FUNCTION_BLOCK ConfigurationManagerC
  (* Standard: 61499-2 *)
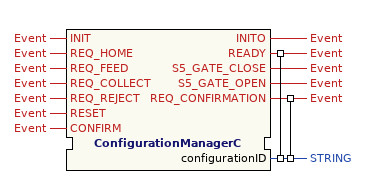
  EVENT_INPUT
    INIT;
    REQ_HOME;
    REQ_FEED;
    REQ_COLLECT;
    REQ_REJECT;
    RESET;
    CONFIRM;
  END_EVENT
  EVENT_OUTPUT
    INITO;
    READY WITH configurationID;
    S5_GATE_CLOSE;
    S5_GATE_OPEN;
    REQ_CONFIRMATION WITH configurationID;
  END_EVENT
  VAR_OUTPUT
    configurationID : STRING;
  END_VAR
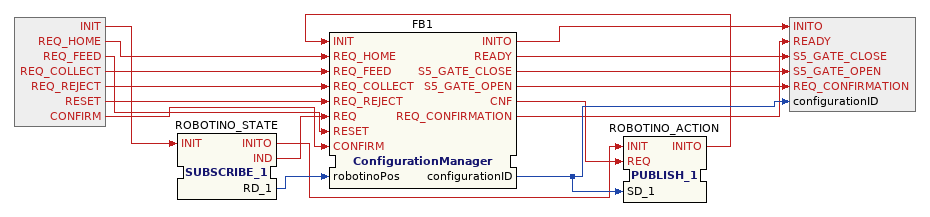
  FBS
    FB1 : ConfigurationManager;
    ROBOTINO_ACTION : PUBLISH_1;
    ROBOTINO_STATE : SUBSCRIBE_1;
  END_FBS
  EVENT_CONNECTIONS
    REQ_HOME TO FB1.REQ_HOME;
    REQ_FEED TO FB1.REQ_FEED;
    REQ_COLLECT TO FB1.REQ_COLLECT;
    REQ_REJECT TO FB1.REQ_REJECT;
    FB1.INITO TO INITO;
    FB1.READY TO READY;
    FB1.S5_GATE_CLOSE TO S5_GATE_CLOSE;
    FB1.S5_GATE_OPEN TO S5_GATE_OPEN;
    ROBOTINO_ACTION.INITO TO FB1.INIT;
    INIT TO ROBOTINO_STATE.INIT;
    RESET TO FB1.RESET;
    FB1.REQ_CONFIRMATION TO REQ_CONFIRMATION;
    CONFIRM TO FB1.CONFIRM;
    ROBOTINO_STATE.INITO TO ROBOTINO_ACTION.INIT;
    ROBOTINO_STATE.IND TO FB1.REQ;
    FB1.CNF TO ROBOTINO_ACTION.REQ;
  END_CONNECTIONS
  DATA_CONNECTIONS
    FB1.configurationID TO ROBOTINO_ACTION.SD_1;
    FB1.configurationID TO configurationID;
    ROBOTINO_STATE.RD_1 TO FB1.robotinoPos;
  END_CONNECTIONS
END_FUNCTION_BLOCK
